{attribute addProperty BoxType "APS4322-5000-0017"}
{attribute addProperty Id "FB_InputsAT %I*FB_Inputs_245CD1AC24643080WcStateAT %I*WcState_F855686C1620InfoDataAT %I*InfoData_7231B2DD80100"}
{attribute addProperty CRC "3520049983"}
{attribute addProperty SizeInBites "2560"}
{attribute addProperty SizeInBytes "320"}
TYPE APS4322_147A8693 :
STRUCT
	{attribute addProperty Name "FB_Inputs"}
	FB_Inputs : FB_Inputs_245CD1AC;
	{attribute addProperty Name "WcState"}
	WcState : WcState_F855686C;
	{attribute addProperty Name "InfoData"}
	InfoData : InfoData_7231B2DD;
END_STRUCT
END_TYPE

(* stored: Version 1.2.0.0, ProductVersion 3.1.4024.9
   DUT APS4322_147A8693: Id {804173a2-f6d6-4fdf-b000-e5251bb88ee6} *)
